{attribute 'GeneratedUsingTerminal: EL1502-0000-0001'}
{attribute addProperty BoxType "EL1502-0000-0001"}
{attribute addProperty Id "CNT_InputsAT %I*CNT_Inputs_147BF88E12CNT_OutputsAT %Q*CNT_Outputs_EB14A6758WcStateAT %I*WcState_9091E0EB2InfoDataAT %I*InfoData_94A18F5E2"}
{attribute addProperty CRC "2663771403"}
{attribute addProperty Size "24"}
TYPE EL1502_9EC5ED0B EXTENDS EtcSlaveTerminalBase_947E5A46 :
STRUCT
	{attribute addProperty Name "CNT_Inputs"}
	CNT_Inputs : CNT_Inputs_147BF88E;
	{attribute addProperty Name "CNT_Outputs"}
	CNT_Outputs : CNT_Outputs_EB14A675;
	{attribute addProperty Name "WcState"}
	WcState : WcState_9091E0EB;
	{attribute addProperty Name "InfoData"}
	InfoData : InfoData_94A18F5E;
END_STRUCT
END_TYPE

(* stored: Version 1.2.0.0, ProductVersion 3.1.4024.9
   DUT EL1502_9EC5ED0B: Id {a21a41bc-45b6-4bf8-8ccf-10480884ee21} *)
